// Mitsubishi GX Works2 project: timer+sequence_1   PLC: Q03UDV

PROGRAM MAIN
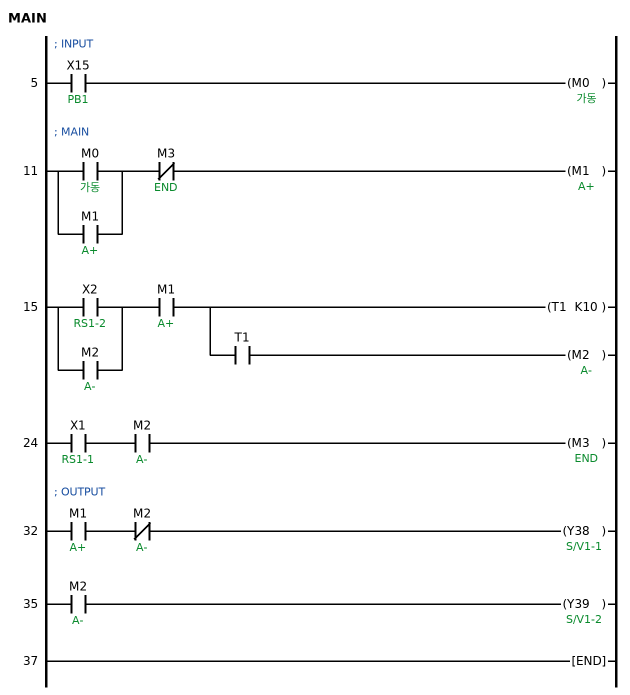
; INPUT
5     LD      X15  ; PB1
      OUT     M0  ; 가동
; MAIN
11    LD      M0  ; 가동
      OR      M1  ; A+
      ANI     M3  ; END
      OUT     M1  ; A+
15    LD      X2  ; RS1-2
      OR      M2  ; A-
      AND     M1  ; A+
      OUT     T1 K10
      AND     T1
      OUT     M2  ; A-
24    LD      X1  ; RS1-1
      AND     M2  ; A-
      OUT     M3  ; END
; OUTPUT
32    LD      M1  ; A+
      ANI     M2  ; A-
      OUT     Y38  ; S/V1-1
35    LD      M2  ; A-
      OUT     Y39  ; S/V1-2
37    END
END_PROGRAM
